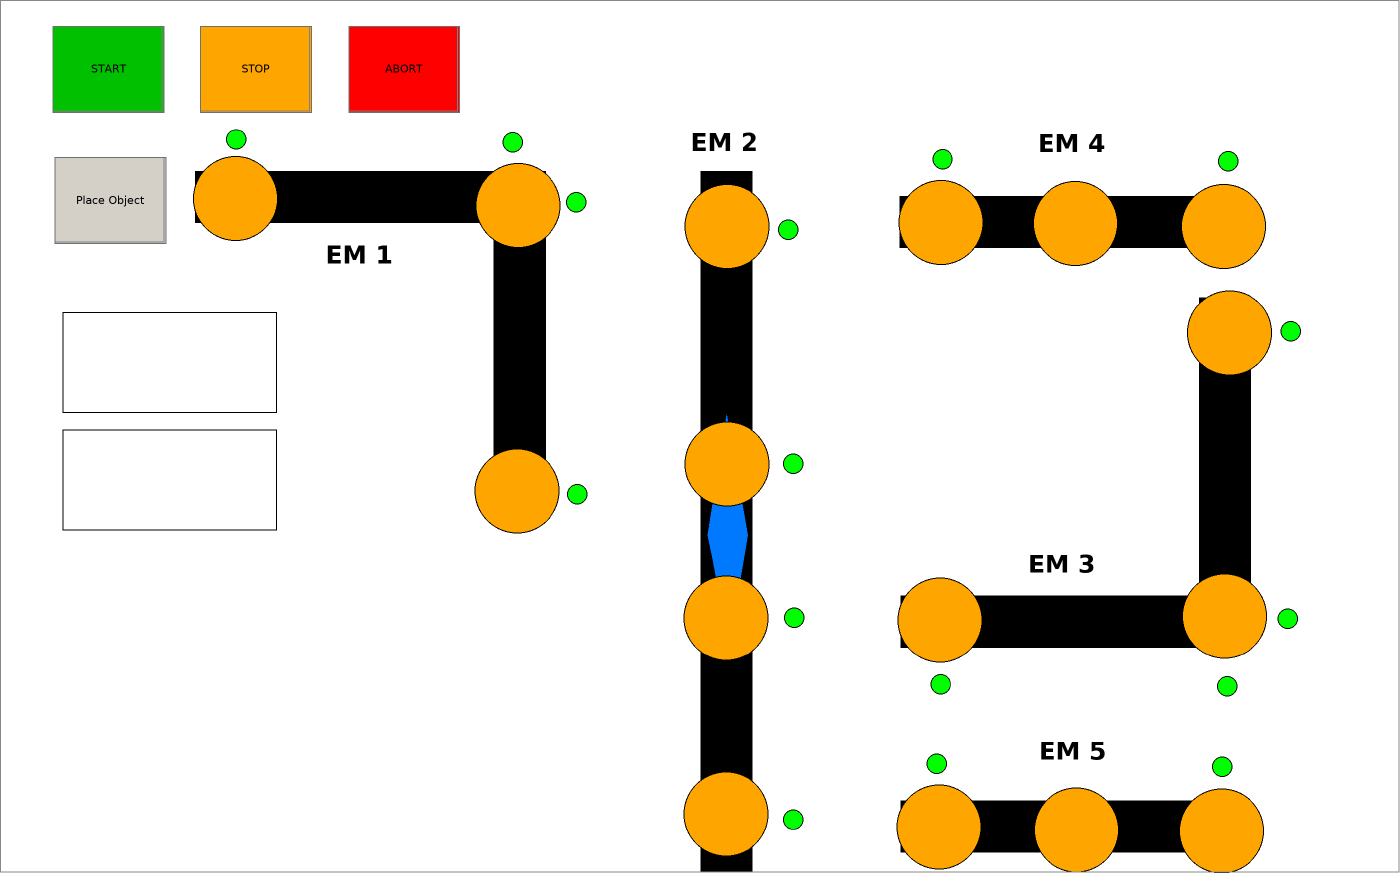
VISUALIZATION VisuPiotrUN  // 1407x878
    Rectangle (196,172 352x52)
    Rectangle (346,322 352x52), angle 90
    Button (55,158 112x87), "Place Object"
        toggle MAIN.cell.PlaceObject
    Ellipse (194,157 85x85), invisible if: NOT (MAIN.fbTaskPiotrUN.em[1].Config.Data.objectSensor AND MAIN.fbTaskPiotrUN.em[1].Config.Data.I[1])
    Button (53,26 112x87), "START"
        toggle MAIN.START
    Button (201,26 112x87), "STOP"
        toggle MAIN.STOP
    Button (350,26 112x87), "ABORT"
        toggle MAIN.ABORT
    Rectangle (378,498 704x52), angle 90
    Ellipse (688,185 85x85), invisible if: NOT (MAIN.fbTaskPiotrUN.em[2].Config.Data.I[3] AND MAIN.fbTaskPiotrUN.em[2].Config.Data.act_pos = 4)
    Ellipse (687,776 85x85), invisible if: NOT (MAIN.fbTaskPiotrUN.em[2].Config.Data.I[3] AND MAIN.fbTaskPiotrUN.em[2].Config.Data.act_pos = 1)
    Rectangle (1055,449 352x52), angle 90
    Rectangle (905,599 352x52)
    Rectangle (904,197 352x52)
    Rectangle (905,805 352x52)
    Ellipse (1187,185 85x85), invisible if: NOT (MAIN.fbTaskPiotrUN.em[4].Config.Data.objectSensor AND MAIN.fbTaskPiotrUN.em[4].Config.Data.I[1])
    Label (286,241 150x30), "EM 1"
    Label (653,128 150x30), "EM 2"
    Label (992,552 150x30), "EM 3"
    Polygon (711,538) (730,417) (751,538) (732,652) (716,562), invisible if: NOT (MAIN.fbTaskPiotrUN.em[2].Config.Data.act_pos = 666)
    Label (1002,129 150x30), "EM 4"
    Label (1003,740 150x30), "EM 5"
    Ellipse (688,424 85x85), invisible if: NOT (MAIN.fbTaskPiotrUN.em[2].Config.Data.I[3] AND MAIN.fbTaskPiotrUN.em[2].Config.Data.act_pos = 3)
    Ellipse (687,579 85x85), invisible if: NOT (MAIN.fbTaskPiotrUN.em[2].Config.Data.I[3] AND MAIN.fbTaskPiotrUN.em[2].Config.Data.act_pos = 2)
    Rectangle (63,432 215x101)
    Rectangle (63,314 215x101)
    Ellipse (505,133 20x20), invisible if: NOT MAIN.fbTaskPiotrUN.em[1].Config.Data.I[2]
    Ellipse (227,130 20x20), invisible if: NOT MAIN.fbTaskPiotrUN.em[1].Config.Data.I[1]
    Ellipse (570,487 20x20), invisible if: NOT MAIN.fbTaskPiotrUN.em[1].Config.Data.I[4]
    Ellipse (569,193 20x20), invisible if: NOT MAIN.fbTaskPiotrUN.em[1].Config.Data.I[3]
    Ellipse (937,150 20x20), invisible if: NOT MAIN.fbTaskPiotrUN.em[4].Config.Data.I[2]
    Ellipse (1224,152 20x20), invisible if: NOT MAIN.fbTaskPiotrUN.em[4].Config.Data.I[1]
    Ellipse (931,758 20x20), invisible if: NOT MAIN.fbTaskPiotrUN.em[5].Config.Data.I[1]
    Ellipse (1218,761 20x20), invisible if: NOT MAIN.fbTaskPiotrUN.em[5].Config.Data.I[2]
    Ellipse (935,678 20x20), invisible if: NOT MAIN.fbTaskPiotrUN.em[3].Config.Data.I[1]
    Ellipse (1223,680 20x20), invisible if: NOT MAIN.fbTaskPiotrUN.em[3].Config.Data.I[2]
    Ellipse (1284,612 20x20), invisible if: NOT MAIN.fbTaskPiotrUN.em[3].Config.Data.I[3]
    Ellipse (1287,323 20x20), invisible if: NOT MAIN.fbTaskPiotrUN.em[3].Config.Data.I[4]
    Ellipse (782,221 20x20), invisible if: NOT (MAIN.fbTaskPiotrUN.em[2].Config.Data.act_pos = 4)
    Ellipse (787,456 20x20), invisible if: NOT (MAIN.fbTaskPiotrUN.em[2].Config.Data.act_pos = 3)
    Ellipse (788,611 20x20), invisible if: NOT (MAIN.fbTaskPiotrUN.em[2].Config.Data.act_pos = 2)
    Ellipse (787,814 20x20), invisible if: NOT ( MAIN.fbTaskPiotrUN.em[2].Config.Data.act_pos = 1)
    Ellipse (478,164 85x85), invisible if: NOT (MAIN.fbTaskPiotrUN.em[1].Config.Data.objectSensor AND MAIN.fbTaskPiotrUN.em[1].Config.Data.I[2] AND MAIN.fbTaskPiotrUN.em[1].Config.Data.I[3])
    Ellipse (477,451 85x85), invisible if: NOT (MAIN.fbTaskPiotrUN.em[1].Config.Data.objectSensor AND MAIN.fbTaskPiotrUN.em[1].Config.Data.I[4])
    Ellipse (1188,577 85x85), invisible if: NOT (MAIN.fbTaskPiotrUN.em[3].Config.Data.objectSensor AND MAIN.fbTaskPiotrUN.em[3].Config.Data.I[2] AND MAIN.fbTaskPiotrUN.em[3].Config.Data.I[3])
    Ellipse (902,581 85x85), invisible if: NOT (MAIN.fbTaskPiotrUN.em[3].Config.Data.objectSensor AND MAIN.fbTaskPiotrUN.em[3].Config.Data.I[1])
    Ellipse (1193,292 85x85), invisible if: NOT (MAIN.fbTaskPiotrUN.em[3].Config.Data.objectSensor AND MAIN.fbTaskPiotrUN.em[3].Config.Data.I[4])
    Ellipse (903,181 85x85), invisible if: NOT (MAIN.fbTaskPiotrUN.em[4].Config.Data.objectSensor AND MAIN.fbTaskPiotrUN.em[4].Config.Data.I[2])
    Ellipse (901,789 85x85), invisible if: NOT (MAIN.fbTaskPiotrUN.em[5].Config.Data.objectSensor AND MAIN.fbTaskPiotrUN.em[5].Config.Data.I[1])
    Ellipse (1185,793 85x85), invisible if: NOT (MAIN.fbTaskPiotrUN.em[5].Config.Data.objectSensor AND MAIN.fbTaskPiotrUN.em[5].Config.Data.I[2])
    Ellipse (1038,182 85x85), invisible if: NOT (MAIN.fbTaskPiotrUN.em[4].Config.Data.objectSensor AND NOT MAIN.fbTaskPiotrUN.em[4].Config.Data.I[2] and not MAIN.fbTaskPiotrUN.em[4].Config.Data.I[1]))
    Ellipse (1039,792 85x85), invisible if: NOT (MAIN.fbTaskPiotrUN.em[5].Config.Data.objectSensor AND NOT MAIN.fbTaskPiotrUN.em[5].Config.Data.I[2] and not MAIN.fbTaskPiotrUN.em[5].Config.Data.I[1]))
END_VISUALIZATION

(* stored: Version 1.1.0.1, ProductVersion 3.1.4024.12
   Visu VisuPiotrUN: Id {563a9b27-6f42-4491-878f-006d45d14b86} *)
